// TIA Portal V16 export
// export: Created 2023-11-14T19:43:15.366354Z, ExportSetting WithDefaults, DisplayName Totally Integrated Automation Portal, DisplayVersion V16, DisplayName TIA Portal Version Control Interface, DisplayVersion V16, DisplayName TIA Portal Openness, DisplayVersion V16, DisplayName SINAMICS Startdrive Advanced, DisplayVersion V16, DisplayName SINAMICS Startdrive G130, G150, S120, S150, SINAMICS MV, S210, DisplayVersion V16, DisplayName SINAMICS Startdrive G110M, G120, G120C, G120D, G120P, DisplayVersion V16, DisplayName STEP 7 Professional, DisplayVersion V16, DisplayName STEP 7 Safety, DisplayVersion V16, DisplayName WinCC Professional, DisplayVersion V16
DATA_BLOCK "CREAR_DB"   // DB7
{ S7_Optimized_Access := 'TRUE' }
VERSION : 0.1
// stored: AutoNumber true, DBAccessibleFromOPCUA true, IsOnlyStoredInLoadMemory false, IsRetainMemResEnabled false, IsWriteProtectedInAS false, MemoryReserve 100
   VAR
      records : UDInt := 17280;
      "name" : String := 'logging';
      id : DWord := 1;
      headers : String := 'HumD11,HumD13,HumD16,TempD11,TempD13,HumMatte,TempMatte';
      data : Struct
         humD11 : Real;
         humD13 : Real;
         humD16 : Real;
         tempD11 : Real;
         tempD13 : Real;
         humMatte : Real;
         tempMatte : Real;
      END_STRUCT;
      done : Bool;
      busy : Bool := true;
      error : Bool;
      status : Word;
   END_VAR
BEGIN
END_DATA_BLOCK
